(* PLC project Tc2_Utilities.WSTRING_TO_UTF8 Demo, tc3-libraries-kb TwinCAT 3.1 *)
(* stored: creationDateTime 2026-05-12T00:00:00, modificationDateTime 2026-05-12T00:00:00 *)

PROGRAM P_Demo_WSTRING_TO_UTF8
  VAR
    wsSrc : WSTRING := "主泵状态";  (* 工业语义：HMI WSTRING 含 Unicode *)
    aUtf8 : ARRAY[0..255] OF BYTE;  (* UTF-8 输出（上云） *)
    bOk : BOOL;  (* 成功 *)
    bConvert : BOOL;  (* 在线触发 *)
  END_VAR

// =============================================================================
// 场景：HMI WSTRING 数据上 OPC UA 云（UA 强制 UTF-8）。
// 价值：比 `WSTRING_TO_STRING2` + `STRING_TO_UTF8` 中转少一次转换。
// 验证步骤：
//   1. 引用 Tc2_Utilities
//   2. 编译 + 登录 + 运行
//   3. 在线写触发位 TRUE，monitor 输出变量
// =============================================================================
IF bConvert THEN
    bOk := WSTRING_TO_UTF8(pDstUTF8    := ADR(aUtf8),
                           pSrcWSTRING := ADR(wsSrc),
                           nDstSize    := SIZEOF(aUtf8));
    bConvert := FALSE;
END_IF;
END_PROGRAM
